Staubli VAL3: GetAxis8Pos.pgx

public program GetAxis8Pos(num& x_nPosition (dimensions=1), num x_nPrecent (dimensions=1))
begin

  dDio["O4_b8RecordPos"]=true
  delay(0.05)
  dDio["O4_b8RecordPos"]=false


  x_nPosition=aioGet(aAio["In4_a8CurPosH"])*power(2,16)+aioGet(aAio["In4_a8CurPosL"])
  x_nPosition=x_nPosition/max(x_nPrecent,0.001)

end
